{attribute 'qualified_only'}
{attribute 'strict'}
TYPE E_ModBusMasterState :
(
	Uninitialized := 0,//0
	Initializing := 10,//10
	Ready	:= 20	,//20
	Running		:= 30,//30
	Stop		:= 200,//200
	Stop_done	:= 210//210
	
);
END_TYPE

(* stored: Version 1.1.0.1, ProductVersion 3.1.4024.12
   DUT E_ModBusMasterState: Id {0f26602f-ad9b-4bf2-8942-c18fb7cf9e70} *)
